{attribute addProperty BoxType "EPP1342-0001-0016"}
{attribute addProperty Id "A_0024_EPP1342_0001_0017A_0024_EPP1342_0001_0017_4205AF082816352"}
{attribute addProperty CRC "3384004469"}
{attribute addProperty SizeInBites "2816"}
{attribute addProperty SizeInBytes "352"}
TYPE A_0023_EPP1342_0001_0016_C9B3CF75 EXTENDS EPP1342_179A0949 :
STRUCT
	{attribute addProperty Name "A_0024_EPP1342_0001_0017"}
	A_0024_EPP1342_0001_0017 : A_0024_EPP1342_0001_0017_4205AF08;
END_STRUCT
END_TYPE

(* stored: Version 1.2.0.0, ProductVersion 3.1.4024.9
   DUT A_0023_EPP1342_0001_0016_C9B3CF75: Id {8abd98ab-f102-4c8a-b738-e7b8d856a80e} *)
